# EPICS autosave request: apps/omegaD5000App/Db/tempSens_chan.req
$(P)$(CHAN):RAW.DESC
$(P)$(CHAN):CAL.B
$(P)$(CHAN):CAL.C
## alarm settings
$(P)$(CHAN)_F.LLSV
$(P)$(CHAN)_F.LOLO
$(P)$(CHAN)_F.LSV
$(P)$(CHAN)_F.LOW
$(P)$(CHAN)_F.HSV
$(P)$(CHAN)_F.HIGH
$(P)$(CHAN)_F.HHSV
$(P)$(CHAN)_F.HIHI
